{attribute addProperty BoxType "EL6201-0000-0017"}
{attribute addProperty Id "Slave_23A_DO0BIT10.125177Slave_23A_DO1BIT10.125178Slave_23A_DO2BIT10.125179Slave_23A_DO3BIT10.125180Slave_23B_DO0BIT10.125181Slave_23B_DO1BIT10.125182Slave_23B_DO2BIT10.125183Slave_23B_DO3BIT10.125184"}
{attribute addProperty CRC "2293011207"}
{attribute addProperty SizeInBites "8"}
{attribute addProperty SizeInBytes "1"}
TYPE Slave_23_Outputs_88AC9307 :
STRUCT
	{attribute addProperty Name "Slave_23A_DO0"}
	Slave_23A_DO0 : BIT;
	{attribute addProperty Name "Slave_23A_DO1"}
	Slave_23A_DO1 : BIT;
	{attribute addProperty Name "Slave_23A_DO2"}
	Slave_23A_DO2 : BIT;
	{attribute addProperty Name "Slave_23A_DO3"}
	Slave_23A_DO3 : BIT;
	{attribute addProperty Name "Slave_23B_DO0"}
	Slave_23B_DO0 : BIT;
	{attribute addProperty Name "Slave_23B_DO1"}
	Slave_23B_DO1 : BIT;
	{attribute addProperty Name "Slave_23B_DO2"}
	Slave_23B_DO2 : BIT;
	{attribute addProperty Name "Slave_23B_DO3"}
	Slave_23B_DO3 : BIT;
END_STRUCT
END_TYPE

(* stored: Version 1.2.0.0, ProductVersion 3.1.4024.9
   DUT Slave_23_Outputs_88AC9307: Id {66d31698-cd13-424b-9d89-a9d755d03dda} *)
